(* CoDeSys 2.3.10.0 project: 2floor.2.pr6 *)
(* Libraries: TcAdsBC.lb6 5.7.02 12:03:02, STANDARD.LB6 5.6.98 12:03:02 *)

(* Global variable list: Global_Variables *)
VAR_GLOBAL
	din1_1	AT %IX52.0:	BOOL;
	din1_2	AT %IX52.1:	BOOL;
	din1_3	AT %IX52.2:	BOOL;
	din1_4	AT %IX52.3:	BOOL;
	din1_5	AT %IX52.4:	BOOL;
	din1_6	AT %IX52.5:	BOOL;
	din1_7	AT %IX52.6:	BOOL;
	din1_8	AT %IX52.7:	BOOL;
	din2_1	AT %IX53.0:	BOOL;
	din2_2	AT %IX53.1:	BOOL;
	din2_3	AT %IX53.2:	BOOL;
	din2_4	AT %IX53.3:	BOOL;
	din2_5	AT %IX53.4:	BOOL;
	din2_6	AT %IX53.5:	BOOL;
	din2_7	AT %IX53.6:	BOOL;
	din2_8	AT %IX53.7:	BOOL;
(*din3_1*)sw_kino_balkon	AT %IX54.0:	BOOL;
(*din3_2*)sw_tambur2		AT %IX54.1:	BOOL;
(*din3_3*)sw_kino1			AT %IX54.2:	BOOL;
(*din3_4*)sw_korydor		AT %IX54.3:	BOOL;
(*din3_5*)sw_kino2			AT %IX54.4:	BOOL;
(*din3_6*)sw_studio1			AT %IX54.5:	BOOL;
(*din3_7*)sw_tambur1		AT %IX54.6:	BOOL;
(*din3_8*)sw_studio2			AT %IX54.7:	BOOL;
(*din4_1*)sw_kabinet1		AT %IX55.0:	BOOL;
	din4_2	AT %IX55.1:	BOOL;
(*din4_3*)sw_kabinet2	AT %IX55.2:	BOOL;
	din4_4	AT %IX55.3:	BOOL;
(*din4_5*)sw_kabinet_balkon	AT %IX55.4:	BOOL;
	din4_6	AT %IX55.5:	BOOL;
(*din4_7*)sw_tambur3		AT %IX55.6:	BOOL;
	din4_8	AT %IX55.7:	BOOL;

(*dout1_1*)balkon_peryla				AT %QX52.0:	BOOL;
(*dout1_2*)kino_l					AT %QX52.1:	BOOL;
(*dout1_3*)balkon_bra				AT %QX52.2:	BOOL;
(*dout1_4*)kabinet_balkon_l			AT %QX52.3:	BOOL;
(*dout1_5*)balkon					AT %QX52.4:	BOOL;
(*dout1_6*)korydor1					AT %QX52.5:	BOOL;
(*dout1_7*)kino_bra					AT %QX52.6:	BOOL;
(*dout1_8*)korydor2					AT %QX52.7:	BOOL;
(*dout2_1*)studio_pidsvitka 			AT %QX53.0:	BOOL;
(*dout2_2*)skhody2_3				AT %QX53.1:	BOOL;
(*dout2_3*)studio_l					AT %QX53.2:	BOOL;
(*dout2_4*)kabinet_pidsvitka_kolo	AT %QX53.3:	BOOL;
(*dout2_5*)kabinet_svitlo				AT %QX53.4:	BOOL;
(*dout2_6*)kabinet_kobra 			AT %QX53.5:	BOOL;
(*dout2_7*)tambur_l					AT %QX53.6:	BOOL;
	stend	AT %QX53.7:	BOOL;
	dout3_1	AT %QX54.0:	BOOL;
(*dout3_2*)fancoil_kabinet_low		AT %QX54.1:	BOOL;
	dout3_3	AT %QX54.2:	BOOL;
(*dout3_4*)fancoil_kabinet_med		AT %QX54.3:	BOOL;
	dout3_5	AT %QX54.4:	BOOL;
	fancoil_kabinet_high				AT %QX54.5:	BOOL;
	dout3_7	AT %QX54.6:	BOOL;
(*dout3_8*)fancoil_kino_low			AT %QX54.7:	BOOL;
(*dout4_1*)fancoil_kino_med			AT %QX55.0:	BOOL;
	dout4_2	AT %QX55.1:	BOOL;
	fancoil_kino_high				AT %QX55.2:	BOOL;
	dout4_4	AT %QX55.3:	BOOL;
	dout4_5	AT %QX55.4:	BOOL;
	dout4_6	AT %QX55.5:	BOOL;
	dout4_7	AT %QX55.6:	BOOL;
	dout4_8	AT %QX55.7:	BOOL;
	dout5_1	AT %QX56.0:	BOOL;
	dout5_2	AT %QX56.1:	BOOL;
	skhody_peryla	AT %QX56.2:	BOOL;
	dout5_4	AT %QX56.3:	BOOL;
	dout5_5	AT %QX56.4:	BOOL;
	dout5_6	AT %QX56.5:	BOOL;
	dout5_7	AT %QX56.6:	BOOL;
	dout5_8	AT %QX56.7:	BOOL;


	klapan_kino 	AT %QB34:	INT;
	klapan_kabinet	AT %QB38:	INT;


	peryla1: BOOL;
	peryla3: BOOL;
	peryla2: BOOL;


END_VAR

(* Global variable list: main *)
VAR_GLOBAL
(*ADS*)
	ads_adr1: STRING:='10.0.5.61.1.1';
	ads_adr2: STRING:='10.0.5.62.1.1';
	ads_adr3: STRING:='10.0.5.63.1.1';

	write_ads: ADSWRITE;
	close_ads:ADSCLOSE;
	read_ads1: ADSREADEX;
	read_ads3: ADSREADEX;

	data3floor: ARRAY[0..3] OF WORD; (*сюди пишуться дані, прочитані з третього поверха*)
	data1floor: ARRAY[0..3] OF WORD; (*сюди пишуться дані, прочитані з третього поверха*)

	skhody2_1 AT %MX0.0: BOOL;
END_VAR

(* Data type *)
TYPE ROOM_HVAC :
STRUCT

	heat_mode:STRING;
	heat_speed:USINT;

	delta_t:SINT;
	t_cur:SINT;
	t_ust:SINT;

	fancoil_speed:SINT;
	klapan:WORD;

	collector1: BOOL;
	collector2: BOOL;
	collector3: BOOL;
	collector4: BOOL;

END_STRUCT
END_TYPE

(* POU MAIN, ST *)
PROGRAM MAIN
VAR

END_VAR
ADS_read;
light;
heat;
END_PROGRAM

(* POU ADS_read, ST *)
PROGRAM ADS_read
VAR
	b_read3: BOOL;
	timer3: TP;
	adsreadtimeout:TIME;
	b_read1: BOOL;
	timer1: TP;
	timeout:TIME;
	errorcounter3: CTU;
	errorcounter1: CTU;
END_VAR
adsreadtimeout:=t#1s;

b_read3:=0;


IF read_ads3.ERR THEN
	timer3.IN:=TRUE;
	b_read3:=FALSE;
ELSE
	timer3.IN:=FALSE;
END_IF

timer3(PT:=adsreadtimeout);
errorcounter3(CU:=timer3.Q);
IF errorcounter3.CV>65534 THEN
	errorcounter3.RESET:=TRUE;
ELSE
	errorcounter3.RESET:=FALSE;
END_IF;
b_read3:= NOT timer3.Q;
IF read_ads3.BUSY THEN
	b_read3:=0;
END_IF

read_ads3(
		NETID:=ads_adr3, (*адреса об'явлена в АДС Глобал*)
		PORT:=801, (*порт першої (основної) рантайм сістем*)
		IDXGRP:=16#4020, (*адресування області %М*)
		IDXOFFS:=4, (*зсув (з якого байта починати читати)*)
		LEN:=8, (*скільки байт прочитати*)
		DESTADDR:=ADR(data3floor), (*розсташування в пам'яті змінної, в яку буде записано те, що прочитали*)
		Read:=b_read3, (*смикаєм за мотузочок, щоб зчитати*)
		TMOUT:=t#2s, (*якщо за секунду не відповість - буде помилка по таймауту*)
	);
timer3.IN:=FALSE;

b_read1:=0;

IF read_ads1.BUSY THEN
	b_read1:=0;
END_IF

IF read_ads1.ERR THEN
	timer1.IN:=TRUE;
ELSE
	timer1.IN:=FALSE;
END_IF

timer1(PT:=adsreadtimeout);
errorcounter1(CU:=timer1.Q);
IF errorcounter1.CV>65534 THEN
	errorcounter1.RESET:=TRUE;
ELSE
	errorcounter1.RESET:=FALSE;
END_IF;

b_read1:= NOT timer1.Q;

IF read_ads1.BUSY THEN
	b_read1:=0;
END_IF

read_ads1(
		NETID:=ads_adr1, (*адреса об'явлена в АДС Глобал*)
		PORT:=800, (*порт першої (основної) рантайм сістем*)
		IDXGRP:=16#4020, (*адресування області %М*)
		IDXOFFS:=0, (*зсув (з якого байта починати читати)*)
		LEN:=1, (*скільки байт прочитати*)
		DESTADDR:=ADR(data1floor), (*розсташування в пам'яті змінної, в яку буде записано те, що прочитали*)
		Read:=b_read1, (*смикаєм за мотузочок, щоб зчитати*)
		TMOUT:=t#2s, (*якщо за секунду не відповість - буде помилка по таймауту*)
	);

timer1.IN:=FALSE;
END_PROGRAM

(* POU light, ST *)
PROGRAM light
VAR
	kino_balkon, kino1, kino2, studio1,studio2, kabinet1, kabinet2, kabinet_balkon, korydor, tambur1, tambur2, tambur3: SWITCH;
	switch_delay: TIME;
	off_delay: TIME;
	sw_skhody2_3:BOOL;
	sw_skhody3_2: BOOL;
	SKHODY2_3R: R_TRIG;
	SKHODY2_3F: F_TRIG;
	skhody1_2: BOOL;
END_VAR
switch_delay:=t#500ms; (*затримка довгого натискання*)
off_delay:=t#3m; (*затримка для відкладеного вимкнення*)

kino_balkon(MODE:='short&long', IN:=sw_kino_balkon,SWITCH_DELAY:=switch_delay, Q_SHORT=>balkon, Q_LONG=>balkon_bra);
balkon_peryla:=kino_balkon.Q_LONG;

kino1(IN:=sw_kino1, SWITCH_DELAY:=switch_delay, Q_SHORT=>kino_l);
kino2(MODE:='short&long', IN:=sw_kino2, SWITCH_DELAY:=switch_delay, Q_SHORT=>kino_bra);
studio1(MODE:='short&long', IN:=sw_studio1, SWITCH_DELAY:=switch_delay, Q_SHORT=>studio_l);
studio2(MODE:='short&long', IN:=sw_studio2, SWITCH_DELAY:=switch_delay, Q_SHORT=>studio_pidsvitka);

korydor(MODE:='short&long', IN:=sw_korydor, SWITCH_DELAY:=switch_delay);
korydor1:=korydor.Q_SHORT;
korydor2:=korydor.Q_SHORT;

kabinet1(MODE:='short&long', IN:=sw_kabinet1, SWITCH_DELAY:=switch_delay, Q_SHORT=>kabinet_svitlo);

kabinet2(MODE:='short&long', IN:=sw_kabinet2, SWITCH_DELAY:=switch_delay);
kabinet_kobra:=kabinet2.Q_SHORT;
kabinet_pidsvitka_kolo:=kabinet2.Q_SHORT;

kabinet_balkon(MODE:='short&long', IN:=sw_kabinet_balkon, SWITCH_DELAY:=switch_delay, Q_SHORT=>kabinet_balkon_l);

tambur2(MODE:='short&long', IN:=sw_tambur2, SWITCH_DELAY:=switch_delay, Q_SHORT=>skhody2_1);
tambur3(MODE:='short&long', IN:=sw_tambur3, SWITCH_DELAY:=switch_delay, Q_SHORT=>stend);

tambur1(MODE:='short&long', IN:=sw_tambur1, SWITCH_DELAY:=switch_delay, Q_SHORT=>sw_skhody2_3);

sw_skhody3_2:=data3floor[0].3;
skhody1_2:=data1floor[0].0;
(*відстежую натискання вимикачів на обох поверхах і перемикаю лампочку по кожному натисненні*)
SKHODY2_3R(CLK:=sw_skhody3_2 XOR sw_skhody2_3);
SKHODY2_3F(CLK:=sw_skhody3_2 XOR sw_skhody2_3);

IF SKHODY2_3R.Q OR SKHODY2_3F.Q THEN
	skhody2_3:=NOT skhody2_3;
	tambur_l:= NOT tambur_l;
END_IF

IF skhody2_3 OR skhody1_2 THEN skhody_peryla:=TRUE;
ELSE skhody_peryla:=FALSE;
END_IF
END_PROGRAM

(* POU Vymykachi/SWITCH, ST *)
FUNCTION_BLOCK SWITCH
VAR_INPUT
	IN:BOOL;
	SWITCH_DELAY:TIME; (*різниця між коротким і довгим натисненням*)
	SHORT_OFF_DELAY, LONG_OFF_DELAY: TIME; (*час затримки вимкнення по короткому та довгому натисненню*)
	MODE:STRING; (*delayed, light, light&vent, short&long, delayed_short&long,  *)
END_VAR
VAR_OUTPUT
	Q_SHORT:BOOL:=FALSE;
	Q_SHORT_D: BOOL;(*вихід для вимкнення із затримкою, вмикається разом із виходом короткого натискання*)
	Q_LONG:BOOL:=FALSE;
	Q_LONG_D:BOOL; (*вихід для вимкнення із затримкою, вмикається разом із виходом довгого натискання*)
END_VAR
VAR
	STAN:BOOL:=FALSE;
	Q_S_fall:F_TRIG; (*ловить задній фронт вихода короткого натискання*)
	Q_L_fall:F_TRIG;(*ловить задній фронт вихода довгого натискання*)
	chas: TIME; (*час доки кнопка натиснена*)

	long: BOOL; (*стає тру, якщо було довге натиснення*)
	short: BOOL; (*стає тру, якщо було коротке натиснення*)
	timer, short_off_delay_timer, long_off_delay_timer: TON; (*таймери: час натискання, час переключення відкладеного виходу по довгому та короткому натисканнях*)
	up: BOOL; (*кнопка натиснена*)

	delay_l, delay_s:BOOL; (*запускати таймери відкладеного вимкнення*)

	turn_off_long: BOOL;
	start_l, start_s:BOOL;
END_VAR
short:=0;
long:=0;
timer(IN:=IN AND STAN, PT:=t#10s);
IF IN AND STAN THEN
	chas:=timer.ET;
	up:=1;
ELSE
up:=0;
END_IF;

IF NOT IN AND NOT STAN THEN
chas:=t#0ms;
END_IF;

IF STAN AND NOT IN THEN
	IF chas <SWITCH_DELAY THEN
		short:=1;
		Q_SHORT:= NOT Q_SHORT;
	END_IF;
	IF chas>=SWITCH_DELAY THEN
		Q_LONG:= NOT Q_LONG;
		long:=1;
	END_IF;
END_IF;

(*затримка вимикання*)
Q_L_fall(CLK:=Q_LONG);
Q_S_fall(CLK:=Q_SHORT);

IF Q_L_FALL.Q THEN
		start_l:=TRUE;
END_IF

IF Q_S_FALL.Q THEN
	start_s:=TRUE;
END_IF

IF MODE='light&vent' THEN
	IF start_s THEN start_l:=start_s; END_IF
END_IF

IF LONG_OFF_DELAY <> t#0ms THEN (*виконувати лише якщо в блок переданий параметр затримки на вимкнення*)

	IF Q_LONG THEN
		Q_LONG_D:=Q_LONG;
	END_IF

	long_off_delay_timer(IN:=start_l, PT:=LONG_OFF_DELAY);

	IF long_off_delay_timer.Q THEN
		Q_LONG_D:=FALSE;
		start_l:=FALSE;
	END_IF

ELSE
	Q_LONG_D:=Q_LONG;
END_IF

IF SHORT_OFF_DELAY <> t#0ms THEN (*виконувати лише якщо в блок переданий параметр затримки на вимкнення*)

	IF Q_SHORT THEN
		Q_SHORT_D:=Q_SHORT;
	END_IF

	short_off_delay_timer(IN:=start_s, PT:=SHORT_OFF_DELAY);

	IF short_off_delay_timer.Q THEN
		Q_SHORT_D:=FALSE;
		start_s:=FALSE;
	END_IF


ELSE
	Q_SHORT_D:=Q_SHORT;
END_IF

IF MODE='delayed' THEN
	Q_LONG:=Q_LONG_D;
	Q_SHORT:=Q_SHORT_D;
END_IF

IF MODE='light' THEN
	Q_SHORT_D:=FALSE;
	Q_LONG:=FALSE;
	Q_LONG_D:=FALSE;
END_IF

IF MODE='short&long' THEN
	Q_SHORT_D:=FALSE;
	Q_LONG_D:=FALSE;
END_IF

IF MODE='light&vent' THEN
	IF NOT Q_SHORT THEN
		Q_LONG:=Q_LONG_D;
	END_IF
END_IF

STAN := IN;
END_FUNCTION_BLOCK

(* POU heat, ST *)
PROGRAM heat
VAR
	fancoil_kino: WORD;
	fancoil_kabinet:  WORD;

END_VAR
	fancoil_kino_low:=data3floor[0].0;
	fancoil_kino_med:=data3floor[0].1;
	fancoil_kino_high:=data3floor[0].2;
	klapan_kino:=data3floor[1];

	fancoil_kabinet_low:=data3floor[2].0;
	fancoil_kabinet_med:=data3floor[2].1;
	fancoil_kabinet_high:=data3floor[2].2;
	klapan_kabinet:=data3floor[3];
END_PROGRAM
